(* IEC 61131-3 sources: CodesysTest/alpha/export/FBs/Components/Bag Delivery/FB_BagDelivery.pou/CommandAcknowledged.prop, 1 file *)

(* ---- Get.pm.st ---- *)
(*#-#-#-#-#-#-#-#-#-#---Declaration---#-#-#-#-#-#-#-#-#-#-#-#-#*)

VAR
END_VAR
(*#-#-#-#-#-#-#-#-#-#---Implementation---#-#-#-#-#-#-#-#-#-#-#-#-#*)

IF _interconnect = BAG_DELIVERY_IC.EIP THEN
	CommandAcknowledged := bagFeedMasterMotor.CommandAcknowledged AND bagFeedRearMotor.CommandAcknowledged;
ELSE
	CommandAcknowledged := bagFeedMasterMotor.CommandAcknowledged;
END_IF
